{attribute 'linkalways'} 
{attribute 'no_explicit_call' := 'This FB is a CLASS and must be accessed using methods or properties'}
{attribute 'enable_dynamic_creation'}
FUNCTION_BLOCK _ETcVnConnectedComponentsAlgorithm EXTENDS EnumDatatypeBase
VAR
	localData : ETcVnConnectedComponentsAlgorithm;
	activeData : REFERENCE TO ETcVnConnectedComponentsAlgorithm;
	enumBaseDatatype : _DINT(localData);
END_VAR

METHOD PRIVATE AddLocalEnumeration
VAR_INPUT
	Enumeration : T_MAXSTRING;
	Value : ETcVnConnectedComponentsAlgorithm;
END_VAR
AddEnumeration(Enumeration, Value);
END_METHOD

PROPERTY PUBLIC Address : PVOID
GET
Address := ADR(activeData);
END_GET
END_PROPERTY

METHOD PUBLIC ClearReference
VAR_INPUT
END_VAR
activeData REF= localData;
SetBaseDatatypeReference();
END_METHOD

METHOD PUBLIC Clone : I_Datatype
VAR
    pClone : POINTER TO _ETcVnConnectedComponentsAlgorithm;
END_VAR
pClone := __NEW(_ETcVnConnectedComponentsAlgorithm(InitialValue := Value));
Clone := pClone^;
END_METHOD

METHOD FB_init : BOOL
VAR_INPUT
	bInitRetains : BOOL; // if TRUE, the retain variables are initialized (warm start / cold start)
	bInCopyCode : BOOL;  // if TRUE, the instance afterwards gets moved into the copy code (online change)
	InitialValue : ETcVnConnectedComponentsAlgorithm;
END_VAR
localData := InitialValue;
AddBaseDatatype(enumBaseDatatype);
ClearReference();

AddLocalEnumeration('TCVN_CCA_WU', ETcVnConnectedComponentsAlgorithm.TCVN_CCA_WU);
AddLocalEnumeration('TCVN_CCA_GRANA', ETcVnConnectedComponentsAlgorithm.TCVN_CCA_GRANA);
END_METHOD

PROPERTY PUBLIC Identifier : T_MAXSTRING
GET
Identifier := 'ETcVnConnectedComponentsAlgorithm';
END_GET
END_PROPERTY

METHOD IsEnumeratorValueEqual : BOOL
VAR_INPUT
	Enumerator : I_KeyValueForwardEnumerator;
END_VAR
VAR
	storedValue : ETcVnConnectedComponentsAlgorithm;
END_VAR
IF NOT Enumerator.TryGet(storedValue) THEN
	RETURN;
END_IF

IsEnumeratorValueEqual := storedValue = activeData;
END_METHOD

METHOD PUBLIC MakeReferenceTo
VAR_INPUT
	ReferenceTarget : REFERENCE TO ETcVnConnectedComponentsAlgorithm;
END_VAR
activeData REF= ReferenceTarget;
SetBaseDatatypeReference();
END_METHOD

METHOD PROTECTED SetBaseDatatypeReference
VAR_INPUT
END_VAR
enumBaseDatatype.MakeReferenceTo(activeData);
END_METHOD

PROPERTY PUBLIC Size : UDINT
GET
Size := SIZEOF(activeData);
END_GET
END_PROPERTY

METHOD TryMakeReferenceTo : BOOL
VAR_INPUT
	Target : I_Datatype;
END_VAR
VAR
	pTargetData : POINTER TO ETcVnConnectedComponentsAlgorithm;
END_VAR
IF NOT IsEquivalentTo(Target) THEN
	RETURN;
END_IF

pTargetData := Target.Address;
activeData REF= pTargetData^;
SetBaseDatatypeReference();
TryMakeReferenceTo := TRUE;
END_METHOD

PROPERTY PUBLIC Value : ETcVnConnectedComponentsAlgorithm
GET
Value := activeData;
END_GET
SET
activeData := Value;
END_SET
END_PROPERTY

END_FUNCTION_BLOCK

(* stored: Version 1.1.0.1, ProductVersion 3.1.4024.13
   POU _ETcVnConnectedComponentsAlgorithm: Id {94b08f52-5259-0029-11bb-6179e92fc307}, SpecialFunc None
   Folder Core: Id {e2698db2-8bae-0bff-26eb-78d22db7d05b}
   Folder Protected: Id {e4b38b0a-401f-0042-2ed4-8ae1d0652dc3}
   Folder Customize: Id {1107d912-6371-0714-2794-eb400501695f}
   Folder Constructor: Id {4862cea3-ccae-0092-337b-931ef608a0a0}
   Folder Private: Id {9035c363-40d5-0e27-12ce-9948b61a8147}
   Folder Protected: Id {86faca90-7108-07c1-2ba8-9413be0d73f6}
   Method AddLocalEnumeration: Id {156f0e76-26f7-07cd-2778-3791ac5dbc84}
   Property Address: Id {4cc4c073-2912-0c52-2116-2003bca60005}
   Get Get: Id {935cb21f-490b-04dc-3fc6-21a2ae9d21e8}
   Method ClearReference: Id {524001af-36e3-01ae-0d09-875f36893ed4}
   Method Clone: Id {23fd32e7-a38c-0bee-2233-23cec9f46dc2}
   Method FB_init: Id {ba6ea52d-bad8-0a7a-2da2-42ed5f8f0960}
   Property Identifier: Id {ea51a171-cdeb-0e5e-37e7-a9676452415b}
   Get Get: Id {0780c089-7141-04de-2e6c-78fa666e72b2}
   Method IsEnumeratorValueEqual: Id {e69c8f74-1c77-0d31-06e6-bdd4a549d9a9}
   Method MakeReferenceTo: Id {350b7051-63e4-0a35-068b-76f8d8b3935f}
   Method SetBaseDatatypeReference: Id {52961e8a-73cf-0055-2270-a0f5c614cebc}
   Property Size: Id {9c0b7f96-16c6-083f-1da9-f4dbcaf8137a}
   Get Get: Id {26bca5f8-ca3b-0b6a-3747-7871639794a7}
   Method TryMakeReferenceTo: Id {227cd649-7a5e-0e1d-3c99-2a416301e026}
   Property Value: Id {09b38df0-b1ef-0293-371e-b627e89e4795}
   Get Get: Id {044d8c41-6c4d-0d55-35c3-5aed11869789}
   Set Set: Id {eac3e1e5-519f-06ca-32f6-d463399d1a25} *)
